// TwinCAT 3 PLC project PLC1
// ProgramVersion: 3.1.4024.0
// libraries:
//   Lib, * (Terza-Automation)
//   Tc2_Standard, * (Beckhoff Automation GmbH)
//   Tc2_System, * (Beckhoff Automation GmbH)
//   Tc2_Utilities, * (Beckhoff Automation GmbH)
//   Tc3_Module, * (Beckhoff Automation GmbH)
//   TcUnit, * (www.tcunit.org)
// project tree:
//   / PlcTask.TcTTO
//   POUs/ AI_OOR.TcPOU, AllCACs.TcPOU, AllCRAHs.TcPOU, AllOtherDis.TcPOU, AllPDUs.TcPOU, All_IO.TcPOU, MAIN.TcPOU, Modbus_RTU.TcPOU, ScaleDP.TcPOU, SystemTime.TcPOU
//   Test/ FB_EventBuffer_Test.TcPOU, PRG_TEST.TcPOU
// real-time tasks:
//   TASK PlcTask: cycle T#10ms, priority 20, ADS port 350
// I/O:
//   DEVICE Device 1 (EtherCAT), AmsNetId 192.168.56.1.2.1
//     Term 1 (EK1100)
// variable links:
//   PLC1 Instance <-> Device 1 (EtherCAT)/Term 1 (EK1100)
//     PlcTask Inputs/GVL_DECI.CouplerStatus <-> InfoData/State
//   PLC1 Instance <-> Device 1 (EtherCAT)/Term 1 (EK1100)/Term 10 (EL1008)
//     PlcTask Inputs/GVL_DECI.Term10Status <-> InfoData/State
//   PLC1 Instance <-> Device 1 (EtherCAT)/Term 1 (EK1100)/Term 11 (EL1008)
//     PlcTask Inputs/GVL_DECI.Term11Status <-> InfoData/State
//   PLC1 Instance <-> Device 1 (EtherCAT)/Term 1 (EK1100)/Term 12 (EL1008)
//     PlcTask Inputs/GVL_DECI.Term12Status <-> InfoData/State
//   PLC1 Instance <-> Device 1 (EtherCAT)/Term 1 (EK1100)/Term 13 (EL1008)
//     PlcTask Inputs/GVL_DECI.Term13Status <-> InfoData/State
//     PlcTask Inputs/MAIN.CRAHs.CRAH_40_02_COM_ALM <-> Channel 8/Input
//     PlcTask Inputs/MAIN.CRAHs.CRAH_40_04_COM_ALM <-> Channel 7/Input
//     PlcTask Inputs/MAIN.CRAHs.CRAH_40_06_COM_ALM <-> Channel 6/Input
//     PlcTask Inputs/MAIN.CRAHs.CRAH_40_14_COM_ALM <-> Channel 5/Input
//     PlcTask Inputs/MAIN.CRAHs.CRAH_40_16_COM_ALM <-> Channel 4/Input
//     PlcTask Inputs/MAIN.CRAHs.CRAH_40_18_COM_ALM <-> Channel 3/Input
//   PLC1 Instance <-> Device 1 (EtherCAT)/Term 1 (EK1100)/Term 14 (EL1008)
//     PlcTask Inputs/GVL_DECI.Term14Status <-> InfoData/State
//     PlcTask Inputs/MAIN.CRAHs.CRAH_40_07_COM_ALM <-> Channel 6/Input
//     PlcTask Inputs/MAIN.CRAHs.CRAH_40_09_COM_ALM <-> Channel 5/Input
//     PlcTask Inputs/MAIN.CRAHs.CRAH_40_11_COM_ALM <-> Channel 4/Input
//     PlcTask Inputs/MAIN.CRAHs.CRAH_40_19_COM_ALM <-> Channel 3/Input
//     PlcTask Inputs/MAIN.CRAHs.CRAH_40_21_COM_ALM <-> Channel 2/Input
//     PlcTask Inputs/MAIN.CRAHs.CRAH_40_23_COM_ALM <-> Channel 1/Input
//     PlcTask Inputs/MAIN.CRAHs.CRAH_40_49_COM_ALM <-> Channel 8/Input
//     PlcTask Inputs/MAIN.CRAHs.CRAH_40_58_COM_ALM <-> Channel 7/Input
//   PLC1 Instance <-> Device 1 (EtherCAT)/Term 1 (EK1100)/Term 15 (EL1008)
//     PlcTask Inputs/GVL_DECI.Term15Status <-> InfoData/State
//     PlcTask Inputs/MAIN.CRAHs.CRAH_40_02_RUN_STS <-> Channel 8/Input
//     PlcTask Inputs/MAIN.CRAHs.CRAH_40_04_RUN_STS <-> Channel 7/Input
//     PlcTask Inputs/MAIN.CRAHs.CRAH_40_06_RUN_STS <-> Channel 6/Input
//     PlcTask Inputs/MAIN.CRAHs.CRAH_40_14_RUN_STS <-> Channel 5/Input
//     PlcTask Inputs/MAIN.CRAHs.CRAH_40_16_RUN_STS <-> Channel 4/Input
//     PlcTask Inputs/MAIN.CRAHs.CRAH_40_18_RUN_STS <-> Channel 3/Input
//     PlcTask Inputs/MAIN.CRAHs.CRAH_40_51_COM_ALM <-> Channel 1/Input
//     PlcTask Inputs/MAIN.CRAHs.CRAH_40_60_COM_ALM <-> Channel 2/Input
//   PLC1 Instance <-> Device 1 (EtherCAT)/Term 1 (EK1100)/Term 16 (EL1008)
//     PlcTask Inputs/GVL_DECI.Term16Status <-> InfoData/State
//     PlcTask Inputs/MAIN.CRAHs.CRAH_40_07_RUN_STS <-> Channel 6/Input
//     PlcTask Inputs/MAIN.CRAHs.CRAH_40_09_RUN_STS <-> Channel 5/Input
//     PlcTask Inputs/MAIN.CRAHs.CRAH_40_11_RUN_STS <-> Channel 4/Input
//     PlcTask Inputs/MAIN.CRAHs.CRAH_40_19_RUN_STS <-> Channel 3/Input
//     PlcTask Inputs/MAIN.CRAHs.CRAH_40_21_RUN_STS <-> Channel 2/Input
//     PlcTask Inputs/MAIN.CRAHs.CRAH_40_23_RUN_STS <-> Channel 1/Input
//     PlcTask Inputs/MAIN.CRAHs.CRAH_40_49_RUN_STS <-> Channel 8/Input
//     PlcTask Inputs/MAIN.CRAHs.CRAH_40_58_RUN_STS <-> Channel 7/Input
//   PLC1 Instance <-> Device 1 (EtherCAT)/Term 1 (EK1100)/Term 17 (EL1008)
//     PlcTask Inputs/GVL_DECI.Term17Status <-> InfoData/State
//     PlcTask Inputs/MAIN.CRAHs.CRAH_40_14_ISOL_1_STS <-> Channel 7/Input
//     PlcTask Inputs/MAIN.CRAHs.CRAH_40_14_ISOL_2_STS <-> Channel 8/Input
//     PlcTask Inputs/MAIN.CRAHs.CRAH_40_16_ISOL_1_STS <-> Channel 5/Input
//     PlcTask Inputs/MAIN.CRAHs.CRAH_40_16_ISOL_2_STS <-> Channel 6/Input
//     PlcTask Inputs/MAIN.CRAHs.CRAH_40_18_ISOL_1_STS <-> Channel 3/Input
//     PlcTask Inputs/MAIN.CRAHs.CRAH_40_18_ISOL_2_STS <-> Channel 4/Input
//     PlcTask Inputs/MAIN.CRAHs.CRAH_40_51_RUN_STS <-> Channel 1/Input
//     PlcTask Inputs/MAIN.CRAHs.CRAH_40_60_RUN_STS <-> Channel 2/Input
//   PLC1 Instance <-> Device 1 (EtherCAT)/Term 1 (EK1100)/Term 18 (EL1008)
//     PlcTask Inputs/GVL_DECI.Term18Status <-> InfoData/State
//     PlcTask Inputs/MAIN.CRAHs.CRAH_40_02_ISOL_1_STS <-> Channel 5/Input
//     PlcTask Inputs/MAIN.CRAHs.CRAH_40_02_ISOL_2_STS <-> Channel 6/Input
//     PlcTask Inputs/MAIN.CRAHs.CRAH_40_04_ISOL_1_STS <-> Channel 3/Input
//     PlcTask Inputs/MAIN.CRAHs.CRAH_40_04_ISOL_2_STS <-> Channel 4/Input
//     PlcTask Inputs/MAIN.CRAHs.CRAH_40_06_ISOL_1_STS <-> Channel 1/Input
//     PlcTask Inputs/MAIN.CRAHs.CRAH_40_06_ISOL_2_STS <-> Channel 2/Input
//     PlcTask Inputs/MAIN.CRAHs.CRAH_40_23_ISOL_1_STS <-> Channel 7/Input
//     PlcTask Inputs/MAIN.CRAHs.CRAH_40_23_ISOL_2_STS <-> Channel 8/Input
//   PLC1 Instance <-> Device 1 (EtherCAT)/Term 1 (EK1100)/Term 19 (EL1008)
//     PlcTask Inputs/GVL_DECI.Term19Status <-> InfoData/State
//     PlcTask Inputs/MAIN.CRAHs.CRAH_40_09_ISOL_1_STS <-> Channel 7/Input
//     PlcTask Inputs/MAIN.CRAHs.CRAH_40_09_ISOL_2_STS <-> Channel 8/Input
//     PlcTask Inputs/MAIN.CRAHs.CRAH_40_11_ISOL_1_STS <-> Channel 5/Input
//     PlcTask Inputs/MAIN.CRAHs.CRAH_40_11_ISOL_2_STS <-> Channel 6/Input
//     PlcTask Inputs/MAIN.CRAHs.CRAH_40_19_ISOL_1_STS <-> Channel 3/Input
//     PlcTask Inputs/MAIN.CRAHs.CRAH_40_19_ISOL_2_STS <-> Channel 4/Input
//     PlcTask Inputs/MAIN.CRAHs.CRAH_40_21_ISOL_1_STS <-> Channel 1/Input
//     PlcTask Inputs/MAIN.CRAHs.CRAH_40_21_ISOL_2_STS <-> Channel 2/Input
//   PLC1 Instance <-> Device 1 (EtherCAT)/Term 1 (EK1100)/Term 2 (EL1008)
//     PlcTask Inputs/GVL_DECI.Term02Status <-> InfoData/State
//     PlcTask Inputs/MAIN.PDUs.PDU17_4_4_1_SPD_STS <-> Channel 1/Input
//   PLC1 Instance <-> Device 1 (EtherCAT)/Term 1 (EK1100)/Term 20 (EL1008)
//     PlcTask Inputs/GVL_DECI.Term20Status <-> InfoData/State
//     PlcTask Inputs/MAIN.CRAHs.CRAH_40_07_ISOL_1_STS <-> Channel 1/Input
//     PlcTask Inputs/MAIN.CRAHs.CRAH_40_07_ISOL_2_STS <-> Channel 2/Input
//     PlcTask Inputs/MAIN.CRAHs.CRAH_40_49_ISOL_1_STS <-> Channel 4/Input
//     PlcTask Inputs/MAIN.CRAHs.CRAH_40_51_ISOL_1_STS <-> Channel 5/Input
//     PlcTask Inputs/MAIN.CRAHs.CRAH_40_58_ISOL_1_STS <-> Channel 3/Input
//     PlcTask Inputs/MAIN.CRAHs.CRAH_40_60_ISOL_1_STS <-> Channel 6/Input
//   PLC1 Instance <-> Device 1 (EtherCAT)/Term 1 (EK1100)/Term 21 (EL1008)
//     PlcTask Inputs/GVL_DECI.Term21Status <-> InfoData/State
//   PLC1 Instance <-> Device 1 (EtherCAT)/Term 1 (EK1100)/Term 22 (EL1008)
//     PlcTask Inputs/GVL_DECI.Term22Status <-> InfoData/State
//   PLC1 Instance <-> Device 1 (EtherCAT)/Term 1 (EK1100)/Term 23 (EL1008)
//     PlcTask Inputs/GVL_DECI.Term23Status <-> InfoData/State
//   PLC1 Instance <-> Device 1 (EtherCAT)/Term 1 (EK1100)/Term 24 (EL1008)
//     PlcTask Inputs/GVL_DECI.Term24Status <-> InfoData/State
//   PLC1 Instance <-> Device 1 (EtherCAT)/Term 1 (EK1100)/Term 25 (EL3058)
//     PlcTask Inputs/GVL_DECI.Term25Status <-> InfoData/State
//   PLC1 Instance <-> Device 1 (EtherCAT)/Term 1 (EK1100)/Term 26 (EL6021)
//     PlcTask Inputs/GVL_DECI.Term26Status <-> InfoData/State
//     PlcTask Inputs/MAIN.ModbusComms.MBComms1.ModbusTerm.InData/D <-> COM TxPDO-Map Inputs/Data In 0
//     PlcTask Inputs/MAIN.ModbusComms.MBComms1.ModbusTerm.InData/D @bit {8..168 step 8} <-> COM TxPDO-Map Inputs/Data In {1..21}  (21 links)
//     PlcTask Outputs/MAIN.ModbusComms.MBComms1.ModbusTerm.OutData/Ctrl <-> COM RxPDO-Map Outputs/Ctrl
//     PlcTask Outputs/MAIN.ModbusComms.MBComms1.ModbusTerm.OutData/D <-> COM RxPDO-Map Outputs/Data Out 0
//     PlcTask Outputs/MAIN.ModbusComms.MBComms1.ModbusTerm.OutData/D @bit {8..168 step 8} <-> COM RxPDO-Map Outputs/Data Out {1..21}  (21 links)
//   PLC1 Instance <-> Device 1 (EtherCAT)/Term 1 (EK1100)/Term 27 (EL6021)
//     PlcTask Inputs/GVL_DECI.Term27Status <-> InfoData/State
//     PlcTask Inputs/MAIN.ModbusComms.MBComms2.ModbusTerm.InData/D <-> COM TxPDO-Map Inputs/Data In 0
//     PlcTask Inputs/MAIN.ModbusComms.MBComms2.ModbusTerm.InData/D @bit {8..168 step 8} <-> COM TxPDO-Map Inputs/Data In {1..21}  (21 links)
//     PlcTask Outputs/MAIN.ModbusComms.MBComms2.ModbusTerm.OutData/Ctrl <-> COM RxPDO-Map Outputs/Ctrl
//     PlcTask Outputs/MAIN.ModbusComms.MBComms2.ModbusTerm.OutData/D <-> COM RxPDO-Map Outputs/Data Out 0
//     PlcTask Outputs/MAIN.ModbusComms.MBComms2.ModbusTerm.OutData/D @bit {8..168 step 8} <-> COM RxPDO-Map Outputs/Data Out {1..21}  (21 links)
//   PLC1 Instance <-> Device 1 (EtherCAT)/Term 1 (EK1100)/Term 28 (EL6021)
//     PlcTask Inputs/GVL_DECI.Term28Status <-> InfoData/State
//     PlcTask Inputs/MAIN.ModbusComms.MBComms3.ModbusTerm.InData/D <-> COM TxPDO-Map Inputs/Data In 0
//     PlcTask Inputs/MAIN.ModbusComms.MBComms3.ModbusTerm.InData/D @bit {8..168 step 8} <-> COM TxPDO-Map Inputs/Data In {1..21}  (21 links)
//     PlcTask Outputs/MAIN.ModbusComms.MBComms3.ModbusTerm.OutData/Ctrl <-> COM RxPDO-Map Outputs/Ctrl
//     PlcTask Outputs/MAIN.ModbusComms.MBComms3.ModbusTerm.OutData/D <-> COM RxPDO-Map Outputs/Data Out 0
//     PlcTask Outputs/MAIN.ModbusComms.MBComms3.ModbusTerm.OutData/D @bit {8..168 step 8} <-> COM RxPDO-Map Outputs/Data Out {1..21}  (21 links)
//   PLC1 Instance <-> Device 1 (EtherCAT)/Term 1 (EK1100)/Term 29 (EL6021)
//     PlcTask Inputs/GVL_DECI.Term29Status <-> InfoData/State
//     PlcTask Inputs/MAIN.ModbusComms.MBComms4.ModbusTerm.InData/D <-> COM TxPDO-Map Inputs/Data In 0
//     PlcTask Inputs/MAIN.ModbusComms.MBComms4.ModbusTerm.InData/D @bit {8..168 step 8} <-> COM TxPDO-Map Inputs/Data In {1..21}  (21 links)
//     PlcTask Outputs/MAIN.ModbusComms.MBComms4.ModbusTerm.OutData/Ctrl <-> COM RxPDO-Map Outputs/Ctrl
//     PlcTask Outputs/MAIN.ModbusComms.MBComms4.ModbusTerm.OutData/D <-> COM RxPDO-Map Outputs/Data Out 0
//     PlcTask Outputs/MAIN.ModbusComms.MBComms4.ModbusTerm.OutData/D @bit {8..168 step 8} <-> COM RxPDO-Map Outputs/Data Out {1..21}  (21 links)
//   PLC1 Instance <-> Device 1 (EtherCAT)/Term 1 (EK1100)/Term 3 (EL1008)
//     PlcTask Inputs/GVL_DECI.Term03Status <-> InfoData/State
//   PLC1 Instance <-> Device 1 (EtherCAT)/Term 1 (EK1100)/Term 30 (EL6021)
//     PlcTask Inputs/GVL_DECI.Term30Status <-> InfoData/State
//     PlcTask Inputs/MAIN.ModbusComms.MBComms5.ModbusTerm.InData/D <-> COM TxPDO-Map Inputs/Data In 0
//     PlcTask Inputs/MAIN.ModbusComms.MBComms5.ModbusTerm.InData/D @bit {8..168 step 8} <-> COM TxPDO-Map Inputs/Data In {1..21}  (21 links)
//     PlcTask Outputs/MAIN.ModbusComms.MBComms5.ModbusTerm.OutData/Ctrl <-> COM RxPDO-Map Outputs/Ctrl
//     PlcTask Outputs/MAIN.ModbusComms.MBComms5.ModbusTerm.OutData/D <-> COM RxPDO-Map Outputs/Data Out 0
//     PlcTask Outputs/MAIN.ModbusComms.MBComms5.ModbusTerm.OutData/D @bit {8..168 step 8} <-> COM RxPDO-Map Outputs/Data Out {1..21}  (21 links)
//   PLC1 Instance <-> Device 1 (EtherCAT)/Term 1 (EK1100)/Term 31 (EL6021)
//     PlcTask Inputs/GVL_DECI.Term31Status <-> InfoData/State
//   PLC1 Instance <-> Device 1 (EtherCAT)/Term 1 (EK1100)/Term 4 (EL1008)
//     PlcTask Inputs/GVL_DECI.Term04Status <-> InfoData/State
//   PLC1 Instance <-> Device 1 (EtherCAT)/Term 1 (EK1100)/Term 5 (EL1008)
//     PlcTask Inputs/GVL_DECI.Term05Status <-> InfoData/State
//   PLC1 Instance <-> Device 1 (EtherCAT)/Term 1 (EK1100)/Term 6 (EL1008)
//     PlcTask Inputs/GVL_DECI.Term06Status <-> InfoData/State
//   PLC1 Instance <-> Device 1 (EtherCAT)/Term 1 (EK1100)/Term 7 (EL1008)
//     PlcTask Inputs/GVL_DECI.Term07Status <-> InfoData/State
//   PLC1 Instance <-> Device 1 (EtherCAT)/Term 1 (EK1100)/Term 8 (EL1008)
//     PlcTask Inputs/GVL_DECI.Term08Status <-> InfoData/State
//   PLC1 Instance <-> Device 1 (EtherCAT)/Term 1 (EK1100)/Term 9 (EL1008)
//     PlcTask Inputs/GVL_DECI.Term09Status <-> InfoData/State

CONFIGURATION PLC1
    RESOURCE PLC ON TwinCAT3
        TASK PlcTask(INTERVAL := T#10ms, PRIORITY := 20);
        PROGRAM MAIN WITH PlcTask : MAIN;
    END_RESOURCE
END_CONFIGURATION

// ---- POUs/MAIN.TcPOU
PROGRAM MAIN
VAR
	PDUs:AllPDUs;
	CRAHs: AllCRAHs;
	IOStatus: All_IO;
	RTUStatus: AllRTUStat;
	CACs: AllCACs;
	IDF: AlllDF;
	OtherDIs: AllOtherDIs;
	EnergyMeters: AllEMeters;
	SystemTimeCall: SystemTime;
	ModbusComms: Modbus_RTU;
	
	bEmpryVar: BOOL;
	fTestFloat: REAL;
	bTestBool: BOOL;
	wTestWord: WORD;
END_VAR


ModbusComms();

CRAHs();
CACs();
PDUs();
IDF();
OtherDIs();
EnergyMeters();

IOStatus();
RTUStatus();

SystemTimeCall();

END_PROGRAM

// ---- POUs/AllPDUs.TcPOU
FUNCTION_BLOCK AllPDUs
VAR
	OnePDU : Lib.OnePDU;
	
	PDU17_4_4_1 : OnePDU;
	
	PDU17_4_4_1_SPD_STS AT %I*: BOOL;
	PDU17_4_4_1_PF_ALM AT %I*: BOOL;
	PDU17_4_4_1_TVOC_BKR_STS AT %I* : BOOL;
	PDU17_4_4_1_TVOC_BKR_TRIP_ALM AT %I* : BOOL;
	PDU17_4_4_1_115_BKR_STS AT %I* : BOOL;
	PDU17_4_4_1_115_BKR_TRIP_ALM AT %I* : BOOL;
	PDU17_4_4_1_125_BKR_STS AT %I* : BOOL;
	PDU17_4_4_1_125_BKR_TRIP_ALM AT %I* : BOOL;
	PDU17_4_4_1_135_BKR_STS AT %I* : BOOL;
	PDU17_4_4_1_135_BKR_TRIP_ALM AT %I* : BOOL;
	PDU17_4_4_1_215_BKR_STS AT %I* : BOOL;
	PDU17_4_4_1_215_BKR_TRIP_ALM AT %I* : BOOL;
	PDU17_4_4_1_225_BKR_STS AT %I* : BOOL;
	PDU17_4_4_1_225_BKR_TRIP_ALM AT %I* : BOOL;
	PDU17_4_4_1_235_BKR_STS AT %I* : BOOL;
	PDU17_4_4_1_235_BKR_TRIP_ALM AT %I* : BOOL;
	
	
	PDU17_4_4_2 : OnePDU;
	
    PDU17_4_4_2_SPD_STS AT %I* : BOOL;
    PDU17_4_4_2_PF_ALM AT %I* : BOOL;
    PDU17_4_4_2_TVOC_BKR_STS AT %I* : BOOL;
    PDU17_4_4_2_TVOC_BKR_TRIP_ALM AT %I* : BOOL;
    PDU17_4_4_2_115_BKR_STS AT %I* : BOOL;
    PDU17_4_4_2_115_BKR_TRIP_ALM AT %I* : BOOL;
    PDU17_4_4_2_125_BKR_STS AT %I* : BOOL;
    PDU17_4_4_2_125_BKR_TRIP_ALM AT %I* : BOOL;
    PDU17_4_4_2_135_BKR_STS AT %I* : BOOL;
    PDU17_4_4_2_135_BKR_TRIP_ALM AT %I* : BOOL;
    PDU17_4_4_2_215_BKR_STS AT %I* : BOOL;
    PDU17_4_4_2_215_BKR_TRIP_ALM AT %I* : BOOL;
    PDU17_4_4_2_225_BKR_STS AT %I* : BOOL;
    PDU17_4_4_2_225_BKR_TRIP_ALM AT %I* : BOOL;
    PDU17_4_4_2_235_BKR_STS AT %I* : BOOL;
    PDU17_4_4_2_235_BKR_TRIP_ALM AT %I* : BOOL;
    PDU17_4_4_2_315_BKR_STS AT %I* : BOOL;
    PDU17_4_4_2_315_BKR_TRIP_ALM AT %I* : BOOL;
    PDU17_4_4_2_325_BKR_STS AT %I* : BOOL;
    PDU17_4_4_2_325_BKR_TRIP_ALM AT %I* : BOOL;
	PDU17_4_4_2_335_BKR_STS AT %I* : BOOL;
    PDU17_4_4_2_335_BKR_TRIP_ALM AT %I* : BOOL;
  

	PDU17_4_4_3 : OnePDU;

	PDU17_4_4_3_SPD_STS AT %I* : BOOL;
    PDU17_4_4_3_PF_ALM AT %I* : BOOL;
    PDU17_4_4_3_TVOC_BKR_STS AT %I* : BOOL;
    PDU17_4_4_3_TVOC_BKR_TRIP_ALM AT %I* : BOOL;
    PDU17_4_4_3_115_BKR_STS AT %I* : BOOL;
    PDU17_4_4_3_115_BKR_TRIP_ALM AT %I* : BOOL;
    PDU17_4_4_3_125_BKR_STS AT %I* : BOOL;
    PDU17_4_4_3_125_BKR_TRIP_ALM AT %I* : BOOL;
    PDU17_4_4_3_135_BKR_STS AT %I* : BOOL;
    PDU17_4_4_3_135_BKR_TRIP_ALM AT %I* : BOOL;
    PDU17_4_4_3_215_BKR_STS AT %I* : BOOL;
    PDU17_4_4_3_215_BKR_TRIP_ALM AT %I* : BOOL;
    PDU17_4_4_3_225_BKR_STS AT %I* : BOOL;
    PDU17_4_4_3_225_BKR_TRIP_ALM AT %I* : BOOL;
    PDU17_4_4_3_235_BKR_STS AT %I* : BOOL;
    PDU17_4_4_3_235_BKR_TRIP_ALM AT %I* : BOOL;
   
   
	PDU17_4_4_4 : OnePDU;
	
	PDU17_4_4_4_SPD_STS AT %I* : BOOL;
    PDU17_4_4_4_PF_ALM AT %I* : BOOL;
    PDU17_4_4_4_TVOC_BKR_STS AT %I* : BOOL;
    PDU17_4_4_4_TVOC_BKR_TRIP_ALM AT %I* : BOOL;
    PDU17_4_4_4_115_BKR_STS AT %I* : BOOL;
    PDU17_4_4_4_115_BKR_TRIP_ALM AT %I* : BOOL;
    PDU17_4_4_4_125_BKR_STS AT %I* : BOOL;
    PDU17_4_4_4_125_BKR_TRIP_ALM AT %I* : BOOL;
    PDU17_4_4_4_135_BKR_STS AT %I* : BOOL;
    PDU17_4_4_4_135_BKR_TRIP_ALM AT %I* : BOOL;
    PDU17_4_4_4_215_BKR_STS AT %I* : BOOL;
    PDU17_4_4_4_215_BKR_TRIP_ALM AT %I* : BOOL;
    PDU17_4_4_4_225_BKR_STS AT %I* : BOOL;
    PDU17_4_4_4_225_BKR_TRIP_ALM AT %I* : BOOL;
    PDU17_4_4_4_235_BKR_STS AT %I* : BOOL;
    PDU17_4_4_4_235_BKR_TRIP_ALM AT %I* : BOOL;
    PDU17_4_4_4_315_BKR_STS AT %I* : BOOL;
    PDU17_4_4_4_315_BKR_TRIP_ALM AT %I* : BOOL;
    PDU17_4_4_4_325_BKR_STS AT %I* : BOOL;
    PDU17_4_4_4_325_BKR_TRIP_ALM AT %I* : BOOL;
	PDU17_4_4_4_335_BKR_STS AT %I* : BOOL;
    PDU17_4_4_4_335_BKR_TRIP_ALM AT %I* : BOOL;

END_VAR


Lib.GVL.nInputCoilIndex      := Lib.GVL_DataHalls.StartInputCoilIndex_PDU;
Lib.GVL.nOutputCoilIndex     := Lib.GVL_DataHalls.StartOutputCoilIndex_PDU;
Lib.GVL.nInputRegisterIndex  := Lib.GVL_DataHalls.StartInputRegisterIndex_PDU;
Lib.GVL.nOutputRegisterIndex := Lib.GVL_DataHalls.StartOutputRegisterIndex_PDU;


PDU17_4_4_1(
	sur_STS         :=PDU17_4_4_1_SPD_STS, 
	phs_ALM         :=PDU17_4_4_1_PF_ALM, 
	sur_phs_offline := Lib.GVL_DECI.Term02Offline, 
	tvoc_BRK_STS    := PDU17_4_4_1_TVOC_BKR_STS , 
	tvoc_BRK_ALM    := PDU17_4_4_1_TVOC_BKR_TRIP_ALM, 
	tvoc_BRK_offline:= Lib.GVL_DECI.Term02Offline, 
	BRK115_POS_STS  := PDU17_4_4_1_115_BKR_STS, 
	BRK115_TRIP_ALM := PDU17_4_4_1_115_BKR_TRIP_ALM, 
	BRK115_offline  := Lib.GVL_DECI.Term02Offline, 
	BRK125_POS_STS  := PDU17_4_4_1_125_BKR_STS, 
	BRK125_TRIP_ALM := PDU17_4_4_1_125_BKR_TRIP_ALM, 
	BRK125_offline  := Lib.GVL_DECI.Term02Offline, 
	BRK135_POS_STS  := PDU17_4_4_1_135_BKR_STS, 
	BRK135_TRIP_ALM := PDU17_4_4_1_135_BKR_TRIP_ALM, 
	BRK135_offline  := Lib.GVL_DECI.Term03Offline, 
	BRK215_POS_STS  := PDU17_4_4_1_215_BKR_STS, 
	BRK215_TRIP_ALM := PDU17_4_4_1_215_BKR_TRIP_ALM, 
	BRK215_offline  := Lib.GVL_DECI.Term03Offline, 
	BRK225_POS_STS  := PDU17_4_4_1_225_BKR_STS, 
	BRK225_TRIP_ALM := PDU17_4_4_1_225_BKR_TRIP_ALM, 
	BRK225_offline  := Lib.GVL_DECI.Term03Offline, 
	BRK235_POS_STS  := PDU17_4_4_1_235_BKR_STS, 
	BRK235_TRIP_ALM := PDU17_4_4_1_235_BKR_TRIP_ALM, 
	BRK235_offline  := Lib.GVL_DECI.Term03Offline, 
	BRK315_POS_STS  := FALSE, 
	BRK315_TRIP_ALM := FALSE, 
	BRK315_offline  := FALSE, 
	BRK325_POS_STS  := FALSE, 
	BRK325_TRIP_ALM := FALSE, 
	BRK325_offline  := FALSE, 
	BRK335_POS_STS  := FALSE, 
	BRK335_TRIP_ALM := FALSE, 
	BRK335_offline  := FALSE, 
	BRK345_POS_STS  := FALSE, 
	BRK345_TRIP_ALM := FALSE, 
	BRK345_offline  := FALSE
);
	
PDU17_4_4_2 (	
	sur_sts := PDU17_4_4_2_SPD_STS,
	phs_ALM := PDU17_4_4_2_PF_ALM,
	sur_phs_offline := Lib.GVL_DECI.Term04Offline,
	tvoc_BRK_STS := PDU17_4_4_2_TVOC_BKR_STS,
	tvoc_BRK_ALM := PDU17_4_4_2_TVOC_BKR_TRIP_ALM,
	tvoc_BRK_offline := Lib.GVL_DECI.Term04Offline,
	BRK115_POS_STS := PDU17_4_4_2_115_BKR_STS,
	BRK115_TRIP_ALM := PDU17_4_4_2_115_BKR_TRIP_ALM,
	BRK115_offline := Lib.GVL_DECI.Term05Offline,
	BRK125_POS_STS := PDU17_4_4_2_125_BKR_STS,
	BRK125_TRIP_ALM := PDU17_4_4_2_125_BKR_TRIP_ALM,
	BRK125_offline := Lib.GVL_DECI.Term05Offline,
	BRK135_POS_STS := PDU17_4_4_2_135_BKR_STS,
	BRK135_TRIP_ALM := PDU17_4_4_2_135_BKR_TRIP_ALM,
	BRK135_offline := Lib.GVL_DECI.Term05Offline,
	BRK215_POS_STS := PDU17_4_4_2_215_BKR_STS,
	BRK215_TRIP_ALM := PDU17_4_4_2_215_BKR_TRIP_ALM,
	BRK215_offline := Lib.GVL_DECI.Term05Offline,
	BRK225_POS_STS := PDU17_4_4_2_225_BKR_STS,
	BRK225_TRIP_ALM := PDU17_4_4_2_225_BKR_TRIP_ALM,
	BRK225_offline := Lib.GVL_DECI.Term06Offline,
	BRK235_POS_STS := PDU17_4_4_2_235_BKR_STS,
	BRK235_TRIP_ALM := PDU17_4_4_2_235_BKR_TRIP_ALM,
	BRK235_offline := Lib.GVL_DECI.Term06Offline,
	BRK315_POS_STS := PDU17_4_4_2_315_BKR_STS,
	BRK315_TRIP_ALM := PDU17_4_4_2_315_BKR_TRIP_ALM,
	BRK315_offline := Lib.GVL_DECI.Term06Offline,
	BRK325_POS_STS := PDU17_4_4_2_325_BKR_STS,
	BRK325_TRIP_ALM := PDU17_4_4_2_325_BKR_TRIP_ALM,
	BRK325_offline := Lib.GVL_DECI.Term06Offline,
    BRK335_POS_STS := PDU17_4_4_2_335_BKR_STS,
	BRK335_TRIP_ALM := PDU17_4_4_2_335_BKR_TRIP_ALM,
	BRK335_offline := Lib.GVL_DECI.Term07Offline,
	BRK345_POS_STS := FALSE,
	BRK345_TRIP_ALM := FALSE,
	BRK345_offline := FALSE
);
	
PDU17_4_4_3 (
	sur_sts := PDU17_4_4_3_SPD_STS,
	phs_ALM := PDU17_4_4_3_PF_ALM,
	sur_phs_offline := Lib.GVL_DECI.Term07Offline,
	tvoc_BRK_STS := PDU17_4_4_3_TVOC_BKR_STS,
	tvoc_BRK_ALM := PDU17_4_4_3_TVOC_BKR_TRIP_ALM,
	tvoc_BRK_offline := Lib.GVL_DECI.Term07Offline,
	BRK115_POS_STS := PDU17_4_4_3_115_BKR_STS,
	BRK115_TRIP_ALM := PDU17_4_4_3_115_BKR_TRIP_ALM,
	BRK115_offline := Lib.GVL_DECI.Term08Offline,
	BRK125_POS_STS := PDU17_4_4_3_125_BKR_STS,
	BRK125_TRIP_ALM := PDU17_4_4_3_125_BKR_TRIP_ALM,
	BRK125_offline := Lib.GVL_DECI.Term08Offline,
	BRK135_POS_STS := PDU17_4_4_3_135_BKR_STS,
	BRK135_TRIP_ALM := PDU17_4_4_3_135_BKR_TRIP_ALM,
	BRK135_offline := Lib.GVL_DECI.Term08Offline,
	BRK215_POS_STS := PDU17_4_4_3_215_BKR_STS,
	BRK215_TRIP_ALM := PDU17_4_4_3_215_BKR_TRIP_ALM,
	BRK215_offline := Lib.GVL_DECI.Term08Offline,
	BRK225_POS_STS := PDU17_4_4_3_225_BKR_STS,
	BRK225_TRIP_ALM := PDU17_4_4_3_225_BKR_TRIP_ALM,
	BRK225_offline := Lib.GVL_DECI.Term09Offline,
	BRK235_POS_STS := PDU17_4_4_3_235_BKR_STS,
	BRK235_TRIP_ALM := PDU17_4_4_3_235_BKR_TRIP_ALM,
	BRK235_offline := Lib.GVL_DECI.Term09Offline,
	BRK315_POS_STS := FALSE,
	BRK315_TRIP_ALM := FALSE,
	BRK315_offline := FALSE,
	BRK325_POS_STS := FALSE,
	BRK325_TRIP_ALM := FALSE,
	BRK325_offline := FALSE,
    BRK335_POS_STS := FALSE,
	BRK335_TRIP_ALM := FALSE,
	BRK335_offline := FALSE,
	BRK345_POS_STS := FALSE,
	BRK345_TRIP_ALM := FALSE,
	BRK345_offline := FALSE
);	

PDU17_4_4_4 ( 
    sur_sts := PDU17_4_4_4_SPD_STS,
	phs_ALM := PDU17_4_4_4_PF_ALM,
	sur_phs_offline := Lib.GVL_DECI.Term10Offline,
	tvoc_BRK_STS := PDU17_4_4_4_TVOC_BKR_STS,
	tvoc_BRK_ALM := PDU17_4_4_4_TVOC_BKR_TRIP_ALM,
	tvoc_BRK_offline := Lib.GVL_DECI.Term10Offline,
	BRK115_POS_STS := PDU17_4_4_4_115_BKR_STS,
	BRK115_TRIP_ALM := PDU17_4_4_4_115_BKR_TRIP_ALM,
	BRK115_offline := Lib.GVL_DECI.Term10Offline,
	BRK125_POS_STS := PDU17_4_4_4_125_BKR_STS,
	BRK125_TRIP_ALM := PDU17_4_4_4_125_BKR_TRIP_ALM,
	BRK125_offline := Lib.GVL_DECI.Term10Offline,
	BRK135_POS_STS := PDU17_4_4_4_135_BKR_STS,
	BRK135_TRIP_ALM := PDU17_4_4_4_135_BKR_TRIP_ALM,
	BRK135_offline := Lib.GVL_DECI.Term11Offline,
	BRK215_POS_STS := PDU17_4_4_4_215_BKR_STS,
	BRK215_TRIP_ALM := PDU17_4_4_4_215_BKR_TRIP_ALM,
	BRK215_offline := Lib.GVL_DECI.Term11Offline,
	BRK225_POS_STS := PDU17_4_4_4_225_BKR_STS,
	BRK225_TRIP_ALM := PDU17_4_4_4_225_BKR_TRIP_ALM,
	BRK225_offline := Lib.GVL_DECI.Term11Offline,
	BRK235_POS_STS := PDU17_4_4_4_235_BKR_STS,
	BRK235_TRIP_ALM := PDU17_4_4_4_235_BKR_TRIP_ALM,
	BRK235_offline := Lib.GVL_DECI.Term11Offline,
	BRK315_POS_STS := PDU17_4_4_4_315_BKR_STS,
	BRK315_TRIP_ALM := PDU17_4_4_4_315_BKR_TRIP_ALM,
	BRK315_offline := Lib.GVL_DECI.Term12Offline,
	BRK325_POS_STS := PDU17_4_4_4_325_BKR_STS,
	BRK325_TRIP_ALM := PDU17_4_4_4_325_BKR_TRIP_ALM,
	BRK325_offline := Lib.GVL_DECI.Term12Offline,
    BRK335_POS_STS := PDU17_4_4_4_335_BKR_STS,
	BRK335_TRIP_ALM := PDU17_4_4_4_335_BKR_TRIP_ALM,
	BRK335_offline := Lib.GVL_DECI.Term12Offline,
	BRK345_POS_STS := FALSE,
	BRK345_TRIP_ALM := FALSE,
	BRK345_offline := FALSE

);

END_FUNCTION_BLOCK

// ---- POUs/AllCRAHs.TcPOU
FUNCTION_BLOCK AllCRAHs
VAR
	OneCRAH : OneCRAH;
	
	CRAH_40_18_COM_ALM AT %I* : BOOL;
	CRAH_40_16_COM_ALM AT %I* : BOOL;
	CRAH_40_14_COM_ALM AT %I* : BOOL;
	CRAH_40_06_COM_ALM AT %I* : BOOL;
	CRAH_40_04_COM_ALM AT %I* : BOOL;
	CRAH_40_02_COM_ALM AT %I* : BOOL;
	CRAH_40_23_COM_ALM AT %I* : BOOL;
	CRAH_40_21_COM_ALM AT %I* : BOOL;
	CRAH_40_19_COM_ALM AT %I* : BOOL;
	CRAH_40_11_COM_ALM AT %I* : BOOL;
	CRAH_40_09_COM_ALM AT %I* : BOOL;
	CRAH_40_07_COM_ALM AT %I* : BOOL;
	CRAH_40_58_COM_ALM AT %I* : BOOL;
	CRAH_40_49_COM_ALM AT %I* : BOOL;
	CRAH_40_51_COM_ALM AT %I* : BOOL;
	CRAH_40_60_COM_ALM AT %I* : BOOL;
	
	CRAH_40_18_RUN_STS AT %I* : BOOL;
	CRAH_40_16_RUN_STS AT %I* : BOOL;
	CRAH_40_14_RUN_STS AT %I* : BOOL;
	CRAH_40_06_RUN_STS AT %I* : BOOL;
	CRAH_40_04_RUN_STS AT %I* : BOOL;
	CRAH_40_02_RUN_STS AT %I* : BOOL;
	CRAH_40_23_RUN_STS AT %I* : BOOL;
	CRAH_40_21_RUN_STS AT %I* : BOOL;
	CRAH_40_19_RUN_STS AT %I* : BOOL;
	CRAH_40_11_RUN_STS AT %I* : BOOL;
	CRAH_40_09_RUN_STS AT %I* : BOOL;
	CRAH_40_07_RUN_STS AT %I* : BOOL;
	CRAH_40_58_RUN_STS AT %I* : BOOL;
	CRAH_40_49_RUN_STS AT %I* : BOOL;
	CRAH_40_51_RUN_STS AT %I* : BOOL;
	CRAH_40_60_RUN_STS AT %I* : BOOL;
	
	
	CRAH_40_18_ISOL_1_STS AT %I* : BOOL;
	CRAH_40_18_ISOL_2_STS AT %I* : BOOL;
	CRAH_40_16_ISOL_1_STS AT %I* : BOOL;
	CRAH_40_16_ISOL_2_STS AT %I* : BOOL;
	CRAH_40_14_ISOL_1_STS AT %I* : BOOL;
	CRAH_40_14_ISOL_2_STS AT %I* : BOOL;
	CRAH_40_06_ISOL_1_STS AT %I* : BOOL;
	CRAH_40_06_ISOL_2_STS AT %I* : BOOL;
	CRAH_40_04_ISOL_1_STS AT %I* : BOOL;
	CRAH_40_04_ISOL_2_STS AT %I* : BOOL;
	CRAH_40_02_ISOL_1_STS AT %I* : BOOL;
	CRAH_40_02_ISOL_2_STS AT %I* : BOOL;
	CRAH_40_23_ISOL_1_STS AT %I* : BOOL;
	CRAH_40_23_ISOL_2_STS AT %I* : BOOL;
	CRAH_40_21_ISOL_1_STS AT %I* : BOOL;
	CRAH_40_21_ISOL_2_STS AT %I* : BOOL;
	CRAH_40_19_ISOL_1_STS AT %I* : BOOL;
	CRAH_40_19_ISOL_2_STS AT %I* : BOOL;
	CRAH_40_11_ISOL_1_STS AT %I* : BOOL;
	CRAH_40_11_ISOL_2_STS AT %I* : BOOL;
	CRAH_40_09_ISOL_1_STS AT %I* : BOOL;
	CRAH_40_09_ISOL_2_STS AT %I* : BOOL;
	CRAH_40_07_ISOL_1_STS AT %I* : BOOL;
	CRAH_40_07_ISOL_2_STS AT %I* : BOOL;
	CRAH_40_58_ISOL_1_STS AT %I* : BOOL;
	CRAH_40_49_ISOL_1_STS AT %I* : BOOL;
	CRAH_40_51_ISOL_1_STS AT %I* : BOOL;
	CRAH_40_60_ISOL_1_STS AT %I* : BOOL;
	
	CRAH_40_18: OneCRAH;
	CRAH_40_16: OneCRAH;
	CRAH_40_14: OneCRAH;
	CRAH_40_06: OneCRAH;
	
	CRAH_40_04: OneCRAH;
	CRAH_40_02: OneCRAH;
	CRAH_40_23: OneCRAH;
	CRAH_40_21: OneCRAH;
	
	CRAH_40_19: OneCRAH;
	CRAH_40_11: OneCRAH;
	CRAH_40_09: OneCRAH;
	CRAH_40_07: OneCRAH;
	
	CRAH_40_58: OneCRAH;
	CRAH_40_49: OneCRAH;
	CRAH_40_51: OneCRAH;
	CRAH_40_60: OneCRAH;
	
	AnyIOOffline: BOOL;
	
END_VAR

Lib.GVL.nInputCoilIndex:= Lib.GVL_DataHalls.StartInputCoilIndex_CRAH;
Lib.GVL.nOutputCoilIndex:= Lib.GVL_DataHalls.StartOutputCoilIndex_CRAH;
Lib.GVL.nInputRegisterIndex:=Lib.GVL_DataHalls.StartInputRegisterIndex_CRAH;
Lib.GVL.nOutputRegisterIndex:=Lib.GVL_DataHalls.StartOutputRegisterIndex_CRAH;

// Crah 40_18
AnyIOOffline:= Lib.GVL_DEci.Term13Offline OR Lib.GVL_DEci.Term15Offline OR Lib.GVL_DEci.Term17Offline;

CRAH_40_18(
	Running:= CRAH_40_18_RUN_STS, 
	Alarm:= CRAH_40_18_COM_ALM, 
	Iso1_1_Sts:= CRAH_40_18_ISOL_1_STS, 
	Iso1_2_Sts:= CRAH_40_18_ISOL_2_STS, 
	Offline:= AnyIOOffline);

// Crah 40_16	
AnyIooffline:= Lib.GVL_DEci.Term13Offline OR Lib.GVL_DEci.Term15Offline OR Lib.GVL_DEci.Term17Offline;

CRAH_40_16(
	Running:= CRAH_40_16_RUN_STS, 
	Alarm:= CRAH_40_16_COM_ALM, 
	Iso1_1_Sts:= CRAH_40_16_ISOL_1_STS, 
	Iso1_2_Sts:= CRAH_40_16_ISOL_2_STS, 
	Offline:= AnyIOOffline);

// Crah 40_14
AnyIooffline:= Lib.GVL_DEci.Term13Offline OR Lib.GVL_DEci.Term15Offline OR Lib.GVL_DEci.Term17Offline;

CRAH_40_14(
	Running:= CRAH_40_14_RUN_STS, 
	Alarm:= CRAH_40_14_COM_ALM, 
	Iso1_1_Sts:= CRAH_40_14_ISOL_1_STS, 
	Iso1_2_Sts:= CRAH_40_14_ISOL_2_STS, 
	Offline:= AnyIOOffline);
	

// Crah 40_06
AnyIooffline:= Lib.GVL_DEci.Term13Offline OR Lib.GVL_DEci.Term15Offline OR Lib.GVL_DEci.Term18Offline;
	
CRAH_40_06(
	Running:= CRAH_40_06_RUN_STS, 
	Alarm:= CRAH_40_06_COM_ALM, 
	Iso1_1_Sts:= CRAH_40_06_ISOL_1_STS, 
	Iso1_2_Sts:= CRAH_40_06_ISOL_2_STS, 
	Offline:= AnyIOOffline);

// Crah 40_04	
AnyIooffline:= Lib.GVL_DEci.Term13Offline OR Lib.GVL_DEci.Term15Offline OR Lib.GVL_DEci.Term18Offline;
	
CRAH_40_04(
	Running:= CRAH_40_04_RUN_STS, 
	Alarm:= CRAH_40_04_COM_ALM, 
	Iso1_1_Sts:= CRAH_40_04_ISOL_1_STS, 
	Iso1_2_Sts:= CRAH_40_04_ISOL_2_STS, 
	Offline:= AnyIOOffline);	
	
// Crah 40_02
AnyIooffline:= Lib.GVL_DEci.Term13Offline OR Lib.GVL_DEci.Term15Offline OR Lib.GVL_DEci.Term18Offline;
	
CRAH_40_02(
	Running:= CRAH_40_02_RUN_STS, 
	Alarm:= CRAH_40_02_COM_ALM, 
	Iso1_1_Sts:= CRAH_40_02_ISOL_1_STS, 
	Iso1_2_Sts:= CRAH_40_02_ISOL_2_STS, 
	Offline:= AnyIOOffline);
	
// Crah 40_02
AnyIooffline:= 	Lib.GVL_DEci.Term14Offline OR Lib.GVL_DEci.Term16Offline OR Lib.GVL_DEci.Term18Offline;
	
CRAH_40_23(
	Running:= CRAH_40_23_RUN_STS, 
	Alarm:= CRAH_40_23_COM_ALM, 
	Iso1_1_Sts:= CRAH_40_23_ISOL_1_STS, 
	Iso1_2_Sts:= CRAH_40_23_ISOL_2_STS, 
	Offline:= AnyIOOffline);

// Crah 40_21	
AnyIooffline:= 	Lib.GVL_DEci.Term14Offline OR Lib.GVL_DEci.Term16Offline OR Lib.GVL_DEci.Term19Offline;
	
CRAH_40_21(
	Running:= CRAH_40_21_RUN_STS, 
	Alarm:= CRAH_40_21_COM_ALM, 
	Iso1_1_Sts:= CRAH_40_21_ISOL_1_STS, 
	Iso1_2_Sts:= CRAH_40_21_ISOL_2_STS, 
	Offline:= AnyIOOffline);
	
// Crah 40_19
AnyIooffline:= Lib.GVL_DEci.Term14Offline OR Lib.GVL_DEci.Term16Offline OR Lib.GVL_DEci.Term19Offline;

CRAH_40_19(
	Running:= CRAH_40_19_RUN_STS, 
	Alarm:= CRAH_40_19_COM_ALM, 
	Iso1_1_Sts:= CRAH_40_19_ISOL_1_STS, 
	Iso1_2_Sts:= CRAH_40_19_ISOL_2_STS, 
	Offline:= AnyIOOffline);
	
// Crah 40_19
AnyIooffline:= Lib.GVL_DEci.Term14Offline OR Lib.GVL_DEci.Term16Offline OR Lib.GVL_DEci.Term19Offline;

CRAH_40_11(
	Running:= CRAH_40_11_RUN_STS, 
	Alarm:= CRAH_40_11_COM_ALM, 
	Iso1_1_Sts:= CRAH_40_11_ISOL_1_STS, 
	Iso1_2_Sts:= CRAH_40_11_ISOL_2_STS, 
	Offline:= AnyIOOffline);	

// Crah 40_09
AnyIooffline:= 	Lib.GVL_DEci.Term14Offline OR Lib.GVL_DEci.Term16Offline OR Lib.GVL_DEci.Term19Offline;
	
CRAH_40_09(
	Running:= CRAH_40_09_RUN_STS, 
	Alarm:= CRAH_40_09_COM_ALM, 
	Iso1_1_Sts:= CRAH_40_09_ISOL_1_STS, 
	Iso1_2_Sts:= CRAH_40_09_ISOL_2_STS, 
	Offline:= AnyIOOffline);
	
// Crah 40_07
AnyIooffline:= 	Lib.GVL_DEci.Term14Offline OR Lib.GVL_DEci.Term16Offline OR Lib.GVL_DEci.Term20Offline;

CRAH_40_07(
	Running:= CRAH_40_07_RUN_STS, 
	Alarm:= CRAH_40_07_COM_ALM, 
	Iso1_1_Sts:= CRAH_40_07_ISOL_1_STS, 
	Iso1_2_Sts:= CRAH_40_07_ISOL_2_STS, 
	Offline:= AnyIOOffline);
	
// Crah 40_58
AnyIooffline:= 	Lib.GVL_DEci.Term14Offline	OR Lib.GVL_DEci.Term16Offline OR Lib.GVL_DEci.Term20Offline;
	
CRAH_40_58(
	Running:= CRAH_40_58_RUN_STS, 
	Alarm:= CRAH_40_58_COM_ALM, 
	Iso1_1_Sts:= CRAH_40_58_ISOL_1_STS, 
	Iso1_2_Sts:= FALSE, 
	Offline:= AnyIOOffline);
	
// Crah 40_49
AnyIooffline:= 	Lib.GVL_DEci.Term14Offline	OR Lib.GVL_DEci.Term16Offline OR Lib.GVL_DEci.Term20Offline;
	
CRAH_40_49(
	Running:= CRAH_40_49_RUN_STS, 
	Alarm:= CRAH_40_49_COM_ALM, 
	Iso1_1_Sts:= CRAH_40_49_ISOL_1_STS, 
	Iso1_2_Sts:= FALSE, 
	Offline:= AnyIOOffline);
	
// Crah 40_51
AnyIooffline:= 	Lib.GVL_DEci.Term15Offline	OR Lib.GVL_DEci.Term17Offline OR Lib.GVL_DEci.Term20Offline;
	
CRAH_40_51(
	Running:= CRAH_40_51_RUN_STS, 
	Alarm:= CRAH_40_51_COM_ALM, 
	Iso1_1_Sts:= CRAH_40_51_ISOL_1_STS, 
	Iso1_2_Sts:= FALSE, 
	Offline:= AnyIOOffline);
	
// Crah 40_60
AnyIooffline:= 	Lib.GVL_DEci.Term15Offline	OR Lib.GVL_DEci.Term17Offline OR Lib.GVL_DEci.Term20Offline;
	
CRAH_40_60(
	Running:= CRAH_40_60_RUN_STS, 
	Alarm:= CRAH_40_60_COM_ALM, 
	Iso1_1_Sts:= CRAH_40_60_ISOL_1_STS, 
	Iso1_2_Sts:= FALSE, 
	Offline:= AnyIOOffline);

END_FUNCTION_BLOCK

// ---- POUs/All_IO.TcPOU
FUNCTION_BLOCK All_IO
VAR_TEMP
	i:INT;
END_VAR


Lib.GVL_DECI.CouplerOffline:= NOT GVL_DECI.CouplerStatus.3;
Lib.GVL_DECI.Term02Offline := NOT GVL_DECI.Term02Status.3;
Lib.GVL_DECI.Term03Offline := NOT GVL_DECI.Term03Status.3;
Lib.GVL_DECI.Term04Offline := NOT GVL_DECI.Term04Status.3;
Lib.GVL_DECI.Term05Offline := NOT GVL_DECI.Term05Status.3;
Lib.GVL_DECI.Term06Offline := NOT GVL_DECI.Term06Status.3;
Lib.GVL_DECI.Term07Offline := NOT GVL_DECI.Term07Status.3;
Lib.GVL_DECI.Term08Offline := NOT GVL_DECI.Term08Status.3;
Lib.GVL_DECI.Term09Offline := NOT GVL_DECI.Term09Status.3;
Lib.GVL_DECI.Term10Offline := NOT GVL_DECI.Term10Status.3;
Lib.GVL_DECI.Term11Offline := NOT GVL_DECI.Term11Status.3;
Lib.GVL_DECI.Term12Offline := NOT GVL_DECI.Term12Status.3;
Lib.GVL_DECI.Term13Offline := NOT GVL_DECI.Term13Status.3;
Lib.GVL_DECI.Term14Offline := NOT GVL_DECI.Term14Status.3;
Lib.GVL_DECI.Term15Offline := NOT GVL_DECI.Term15Status.3;
Lib.GVL_DECI.Term16Offline := NOT GVL_DECI.Term16Status.3;
Lib.GVL_DECI.Term17Offline := NOT GVL_DECI.Term17Status.3;
Lib.GVL_DECI.Term18Offline := NOT GVL_DECI.Term18Status.3;
Lib.GVL_DECI.Term19Offline := NOT GVL_DECI.Term19Status.3;
Lib.GVL_DECI.Term20Offline := NOT GVL_DECI.Term20Status.3;
Lib.GVL_DECI.Term21Offline := NOT GVL_DECI.Term21Status.3;
Lib.GVL_DECI.Term22Offline := NOT GVL_DECI.Term22Status.3;
Lib.GVL_DECI.Term23Offline := NOT GVL_DECI.Term23Status.3;
Lib.GVL_DECI.Term24Offline := NOT GVL_DECI.Term24Status.3;
Lib.GVL_DECI.Term25Offline := NOT GVL_DECI.Term25Status.3;
Lib.GVL_DECI.Term26Offline := NOT GVL_DECI.Term26Status.3;
Lib.GVL_DECI.Term27Offline := NOT GVL_DECI.Term27Status.3;
Lib.GVL_DECI.Term28Offline := NOT GVL_DECI.Term28Status.3;
Lib.GVL_DECI.Term29Offline := NOT GVL_DECI.Term29Status.3;
Lib.GVL_DECI.Term30Offline := NOT GVL_DECI.Term30Status.3;
Lib.GVL_DECI.Term31Offline := NOT GVL_DECI.Term31Status.3;

Lib.GVL.nInputCoilIndex     := Lib.GVL_DataHalls.StartInputCoilIndex_IO;
Lib.GVL.nOutputCoilIndex    := Lib.GVL_DataHalls.StartOutputCoilIndex_IO;
Lib.GVL.nInputRegisterIndex := Lib.GVL_DataHalls.StartInputRegisterIndex_IO;
Lib.GVL.nOutputRegisterIndex:= Lib.GVL_DataHalls.StartOutputRegisterIndex_IO;

i:=Lib.GVL.nInputCoilIndex ;

Lib.GVL.mb_Input_Coils[i+0] := Lib.GVL_DECI.CouplerOffline;
Lib.GVL.mb_Input_Coils[i+1] := Lib.GVL_DECI.Term02Offline;
Lib.GVL.mb_Input_Coils[i+2] := Lib.GVL_DECI.Term03Offline;
Lib.GVL.mb_Input_Coils[i+3] := Lib.GVL_DECI.Term04Offline;
Lib.GVL.mb_Input_Coils[i+4] := Lib.GVL_DECI.Term05Offline;
Lib.GVL.mb_Input_Coils[i+5] := Lib.GVL_DECI.Term06Offline;
Lib.GVL.mb_Input_Coils[i+6] := Lib.GVL_DECI.Term07Offline;
Lib.GVL.mb_Input_Coils[i+7] := Lib.GVL_DECI.Term08Offline;
Lib.GVL.mb_Input_Coils[i+8] := Lib.GVL_DECI.Term09Offline;
Lib.GVL.mb_Input_Coils[i+9] := Lib.GVL_DECI.Term10Offline;
Lib.GVL.mb_Input_Coils[i+10]:= Lib.GVL_DECI.Term11Offline;
Lib.GVL.mb_Input_Coils[i+11]:= Lib.GVL_DECI.Term12Offline;
Lib.GVL.mb_Input_Coils[i+12]:= Lib.GVL_DECI.Term13Offline;
Lib.GVL.mb_Input_Coils[i+13]:= Lib.GVL_DECI.Term14Offline;
Lib.GVL.mb_Input_Coils[i+14]:= Lib.GVL_DECI.Term15Offline;
Lib.GVL.mb_Input_Coils[i+15]:= Lib.GVL_DECI.Term16Offline;
Lib.GVL.mb_Input_Coils[i+16]:= Lib.GVL_DECI.Term17Offline;
Lib.GVL.mb_Input_Coils[i+17]:= Lib.GVL_DECI.Term18Offline;
Lib.GVL.mb_Input_Coils[i+18]:= Lib.GVL_DECI.Term19Offline;
Lib.GVL.mb_Input_Coils[i+19]:= Lib.GVL_DECI.Term20Offline;
Lib.GVL.mb_Input_Coils[i+20]:= Lib.GVL_DECI.Term21Offline;
Lib.GVL.mb_Input_Coils[i+21]:= Lib.GVL_DECI.Term22Offline;
Lib.GVL.mb_Input_Coils[i+22]:= Lib.GVL_DECI.Term23Offline;
Lib.GVL.mb_Input_Coils[i+23]:= Lib.GVL_DECI.Term24Offline;
Lib.GVL.mb_Input_Coils[i+24]:= Lib.GVL_DECI.Term25Offline;
Lib.GVL.mb_Input_Coils[i+25]:= Lib.GVL_DECI.Term26Offline;
Lib.GVL.mb_Input_Coils[i+26]:= Lib.GVL_DECI.Term27Offline;
Lib.GVL.mb_Input_Coils[i+27]:= Lib.GVL_DECI.Term28Offline;
Lib.GVL.mb_Input_Coils[i+28]:= Lib.GVL_DECI.Term29Offline;
Lib.GVL.mb_Input_Coils[i+29]:= Lib.GVL_DECI.Term30Offline;
Lib.GVL.mb_Input_Coils[i+30]:= Lib.GVL_DECI.Term31Offline;
Lib.GVL.mb_Input_Coils[i+31]:= FALSE;
Lib.GVL.mb_Input_Coils[i+32]:= FALSE;
Lib.GVL.mb_Input_Coils[i+33]:= FALSE;
Lib.GVL.mb_Input_Coils[i+34]:= FALSE;
Lib.GVL.mb_Input_Coils[i+35]:= FALSE;
Lib.GVL.mb_Input_Coils[i+36]:= FALSE;

END_FUNCTION_BLOCK

// ---- POUs/AllCACs.TcPOU
FUNCTION_BLOCK AllCACs
VAR_INPUT
END_VAR
VAR_OUTPUT
END_VAR
VAR
END_VAR

END_FUNCTION_BLOCK

// ---- POUs/AllOtherDis.TcPOU
FUNCTION_BLOCK AllOtherDis
VAR
	OneDi: Lib.OneDI;
	
	PSU1_ALM AT %I* : BOOL;
	PSU2_ALM AT %I* : BOOL;
	FAP_PNL_ALM AT %I* : BOOL;
	FAP_LOOP_ALM AT %I* : BOOL;
	Telco_ASD_A_PNL_ALM AT %I* : BOOL;
	Telco_ASD_B_PNL_ALM AT %I* : BOOL;
	DH_ASD_PNL_ALM AT %I* : BOOL;
	
	
	PSU1_Healthy: OneDI;
	PSU2_Healthy: OneDI;
	FAP_Healthy: OneDI;
	FAPL_Healthy: OneDI;
	TelcoSDP_A_Healthy: OneDI;
	TelcoSDP_B_Healthy: OneDI;
	DHSDP_Healthy: OneDI;
	
	UPS_BAT_LOW_ALM AT %I* : BOOL;
	UPS_BAT_MODE    AT %I* : BOOL;
	
	UPS_BatLow: OneDI;
	UPS_BatMode: OneDI;
	

END_VAR


Lib.GVL.nInputCoilIndex     := Lib.GVL_DataHalls.StartInputCoilIndex_OtherDIs;
Lib.GVL.nOutputCoilIndex    := Lib.GVL_DataHalls.StartOutputCoilIndex_OtherDIs;
Lib.GVL.nInputRegisterIndex := Lib.GVL_DataHalls.StartInputRegisterIndex_OtherDIs;
Lib.GVL.nOutputRegisterIndex:= Lib.GVL_DataHalls.StartOutputRegisterIndex_OtherDIs;


PSU1_Healthy(Value:=PSU1_ALM,
			 Offline:= Lib.GVL_DECI.Term13Offline);
			 
PSU2_Healthy(Value:=PSU2_ALM,
			 Offline:= Lib.GVL_DECI.Term13Offline);	
		 
FAP_Healthy(Value:= FAP_PNL_ALM,
			Offline:= Lib.GVL_DECI.Term20Offline);
			
FAPL_Healthy(Value:= FAP_LOOP_ALM,
			 Offline:= Lib.GVL_DECI.Term20Offline);
			 
TelcoSDP_A_Healthy(Value:= Telco_ASD_A_PNL_ALM,
				   Offline:= Lib.GVL_DECI.Term21Offline );

TelcoSDP_B_Healthy(Value:= Telco_ASD_B_PNL_ALM,
				   Offline:= Lib.GVL_DECI.Term21Offline);

DHSDP_Healthy(Value:= DH_ASD_PNL_ALM,
			  Offline:= Lib.GVL_DECI.Term21Offline);
			  
			  
UPS_BatLow(Value:= UPS_BAT_LOW_ALM,
		   Offline:=Lib.GVL_DECI.Term21Offline);
		   
		   
		   
		   // sdf sdf
		   

UPS_BatMode(Value:= UPS_BAT_MODE,
			Offline:=Lib.GVL_DECI.Term21Offline);

END_FUNCTION_BLOCK

// ---- POUs/SystemTime.TcPOU
FUNCTION_BLOCK SystemTime
VAR_INPUT
END_VAR
VAR_OUTPUT
END_VAR
VAR
END_VAR


fbGetLocalSystemTime(
	sNetID:= , 
	bEnable:= TRUE, 
	dwCycle:= 1, 
	dwOpt:= , 
	tTimeout:= , 
	bValid=> , 
	systemTime=> , 
	tzID=> );

Lib.GVL_DECI.sSystemDateTime :=  SYSTEMTIME_TO_STRING(Lib.GVL_DECI.fbGetLocalSystemTime.systemTime);
Lib.GVL_DECI.sSystemDate:= MID(STR:=Lib.GVL_DECI.sSystemDateTime, LEN:=10, POS:=1);
Lib.GVL_DECI.sSystemTime:= MID(STR:=Lib.GVL_DECI.sSystemDateTime, LEN:=8, POS:=12);

END_FUNCTION_BLOCK

// ---- POUs/Modbus_RTU.TcPOU
FUNCTION_BLOCK Modbus_RTU
VAR
	MBComms1: ModbusRTU_THT;
	MBComms2: ModbusRTU_THT;
	MBComms3: ModbusRTU_THT;
	MBComms4: ModbusRTU_THT;
	MBComms5: Modbus_EM;

END_VAR


MBComms1(MB_FirstUnitID:= 1, MB_LastUnitID:= 4);
MBComms2(MB_FirstUnitID:= 5, MB_LastUnitID:= 8);
MBComms3(MB_FirstUnitID:= 9, MB_LastUnitID:= 12);
MBComms4(MB_FirstUnitID:= 13, MB_LastUnitID:= 14);
MBComms5(MB_FirstUnitID:= 15, MB_LastUnitID:= 16);

END_FUNCTION_BLOCK

// ---- POUs/AI_OOR.TcPOU
FUNCTION AI_OOR : BOOL
VAR_INPUT
	Status:WORD;
END_VAR

// calculate whether the status for an analog input is indicating an error
// the error bit is the 7th bit of the status word
// access to bits is base 0, so the 7th bit is accessed with index 6

AI_OOR:= Status.6;

END_FUNCTION

// ---- POUs/ScaleDP.TcPOU
FUNCTION ScaleDP : real
VAR_INPUT
	
END_VAR
VAR
END_VAR

// Raw value of 0 to 32767 scales to -50 to +50

//ScaleDP:=

END_FUNCTION

// ---- Test/FB_EventBuffer_Test.TcPOU
FUNCTION_BLOCK FB_EventBuffer_Test EXTENDS FB_TestSuite
VAR
	

END_VAR



AddThreeEvents();

METHOD PRIVATE AddThreeEvents
VAR
	
	bOk: BOOL;
	nFoo:UDINT;
	
	
END_VAR

Test("AddThreeEvents");


	bOk:=FALSE;

	AssertTrue(Condition:=bOk, Message:="bool variable");
	
	
	nFoo:=1;
	
	
	AssertEquals_UDINT(Expected :=1, Actual:=nFoo, Message:="udint variable");
	
	
	

TEST_FINISHED();
END_METHOD

END_FUNCTION_BLOCK

// ---- Test/PRG_TEST.TcPOU
PROGRAM PRG_TEST
VAR
	foo:FB_EventBuffer_Test;	



END_VAR

TcUnit.RUN();

END_PROGRAM
